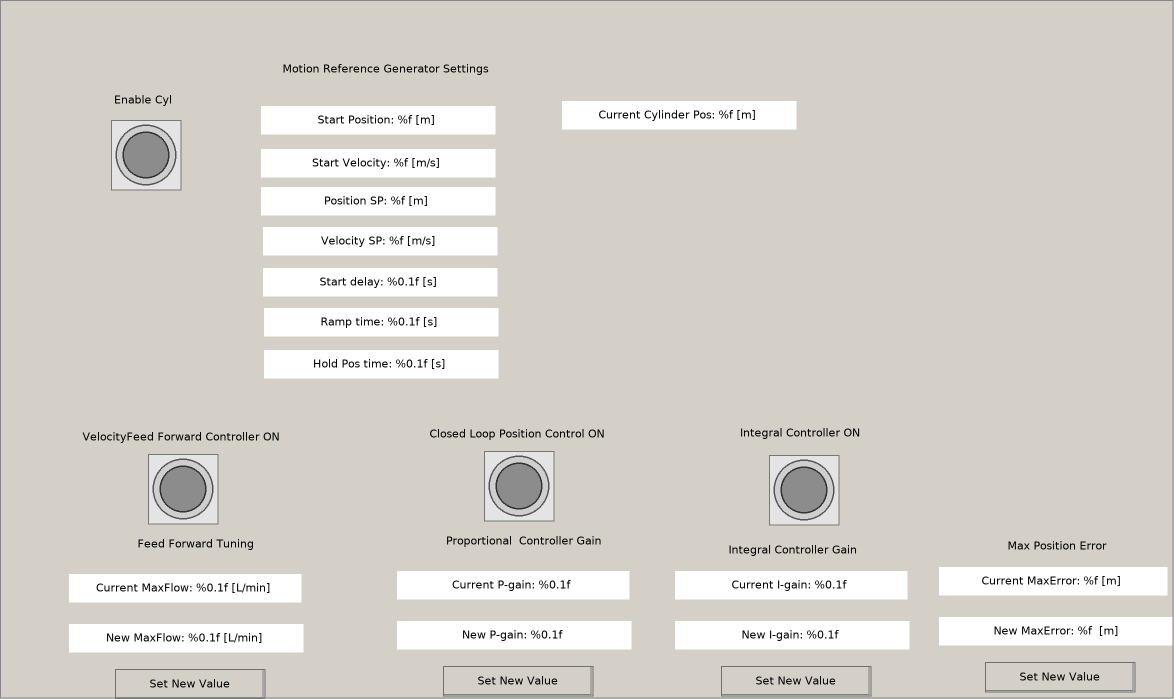
VISUALIZATION Cylinder  // 1174x699
    Label (68,85 150x30), "Enable Cyl"
    PushSwitch (111,120 70x70), variable: G_Hmi.bCylEnable, behaviour: TOGGLE, style: Switch-PushSwitch-Gray
    Label (240,54 291x30), "Motion Reference Generator Settings"
    Textfield (260,105 236x30), "Start Position: %f [m]", text variable: G_Hmi.stMotionReferenceGeneratorSettingsCylinder.fStartPosition_m
        OnMouseDown: write the text variable via Default, min 0, max 0.5
    Textfield (260,148 236x30), "Start Velocity: %f [m/s]", text variable: G_Hmi.stMotionReferenceGeneratorSettingsCylinder.fStartVelocity_m
        OnMouseDown: write the text variable via Default, min 0, max 0.05
    Textfield (260,186 236x30), "Position SP: %f [m]", text variable: G_Hmi.stMotionReferenceGeneratorSettingsCylinder.fPositionSetpoint_ms
        OnMouseDown: write the text variable via Default, min 0, max 0.45
    Textfield (262,226 236x30), "Velocity SP: %f [m/s]", text variable: G_Hmi.stMotionReferenceGeneratorSettingsCylinder.fVelocitySetpoint_m
        OnMouseDown: write the text variable via Default, min 0, max 0.05
    Textfield (262,267 236x30), "Start delay: %0.1f [s]", text variable: G_Hmi.stMotionReferenceGeneratorSettingsCylinder.fTimeBeforeStarting_s
        OnMouseDown: write the text variable via Default, min 0, max 10
    Textfield (263,307 236x30), "Ramp time: %0.1f [s]", text variable: G_Hmi.stMotionReferenceGeneratorSettingsCylinder.fRampTime_s
        OnMouseDown: write the text variable via Default, min 0, max 10
    Textfield (263,349 236x30), "Hold Pos time: %0.1f [s]", text variable: G_Hmi.stMotionReferenceGeneratorSettingsCylinder.fHoldPositionTime_s
        OnMouseDown: write the text variable via Default, min 0, max 10
    Textfield (561,100 236x30), "Current Cylinder Pos: %f [m]", text variable: G_Sensors.fPositionCylPiston
        OnMouseDown: write the text variable via Default, min 0, max 0.5
    Button (443,666 150x30), "Set New Value"
        tap G_Hmi.stModifyAutomaticControlSettingsCylinder.bSetNewProportionalGain
    Textfield (396,570 234x30), "Current P-gain: %0.1f", text variable: G_Parameters.stParam.stClosedLoopControlSettingsCylinder.fProportionalGain
    Textfield (396,620 236x30), "New P-gain: %0.1f", text variable: G_Hmi.stModifyAutomaticControlSettingsCylinder.fNewProportionalGain
        OnMouseDown: write the text variable via Default
    Label (441,526 166x30), "Proportional Controller Gain"
    Button (721,666 150x30), "Set New Value"
        tap G_Hmi.stModifyAutomaticControlSettingsCylinder.bSetNewIntegralGain
    Textfield (674,570 234x30), "Current I-gain: %0.1f", text variable: G_Parameters.stParam.stClosedLoopControlSettingsCylinder.fIntegralGain
    Textfield (674,620 236x30), "New I-gain: %0.1f", text variable: G_Hmi.stModifyAutomaticControlSettingsCylinder.fNewIntegralGain
        OnMouseDown: write the text variable via Default
    Label (718,535 150x30), "Integral Controller Gain"
    PushSwitch (769,455 70x70), variable: G_Hmi.stAutomaticControlSettingsCylinder.bEnableIntegralController, behaviour: TOGGLE, style: Switch-PushSwitch-Gray
    Label (717,418 166x30), "Integral Controller ON"
    Label (391,419 252x30), "Closed Loop Position Control ON"
    PushSwitch (484,451 70x70), variable: G_Hmi.stAutomaticControlSettingsCylinder.bEnableClosedLoopPositionControl, behaviour: TOGGLE, style: Switch-PushSwitch-Gray
    Label (55,422 252x30), "VelocityFeed Forward Controller ON"
    PushSwitch (148,454 70x70), variable: G_Hmi.stAutomaticControlSettingsCylinder.bEnableVelocityFeedForwardControl, behaviour: TOGGLE, style: Switch-PushSwitch-Gray
    Button (115,669 150x30), "Set New Value"
        tap G_Hmi.stModifyAutomaticControlSettingsCylinder.bSetNewMaxFlowCapacity p1329445385=TRUE
    Textfield (68,573 234x30), "Current MaxFlow: %0.1f [L/min]", text variable: G_Parameters.stParam.stOpenLoopControlSettingsCylinder.fMaxFlowCapacity
    Textfield (68,623 236x30), "New MaxFlow: %0.1f [L/min]", text variable: G_Hmi.stModifyAutomaticControlSettingsCylinder.fNewMaxFlowCapacity
        OnMouseDown: write the text variable via Default, min 0.0001, max 100
    Label (113,529 166x30), "Feed Forward Tuning"
    Button (985,662 150x30), "Set New Value"
        tap G_Hmi.stModifyAutomaticControlSettingsCylinder.bSetNewMaxPositionError
    Textfield (938,566 230x30), "Current MaxError: %f [m]", text variable: G_Parameters.stParam.stClosedLoopControlSettingsCylinder.fMaxPositionError
    Textfield (938,616 236x30), "New MaxError: %f [m]", text variable: G_Hmi.stModifyAutomaticControlSettingsCylinder.fNewMaxPositionError
        OnMouseDown: write the text variable via Default
    Label (982,531 150x30), "Max Position Error"
END_VISUALIZATION

(* stored: Version 1.1.0.1, ProductVersion 3.1.4024.11
   Visu Cylinder: Id {0f33c311-d340-48cc-b080-c178a6a4a97e} *)
